FUNCTION_BLOCK Controller
  (* Standard: 61499-2 *)
  (* Version 0.1, 2015-00-21, Th?o, PC_THEO *)
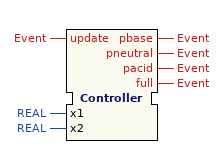
  EVENT_INPUT
    update;
  END_EVENT
  EVENT_OUTPUT
    pbase;
    pneutral;
    pacid;
    full;
  END_EVENT
  VAR_INPUT
    x1 : REAL;
    x2 : REAL;
  END_VAR
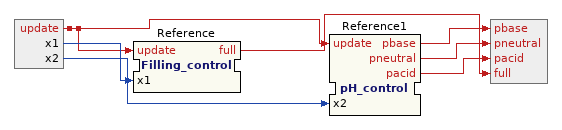
  FBS
    Reference : Filling_control;
    Reference1 : pH_control;
  END_FBS
  EVENT_CONNECTIONS
    update TO Reference.update;
    update TO Reference1.update;
    Reference1.pbase TO pbase;
    Reference1.pneutral TO pneutral;
    Reference1.pacid TO pacid;
    Reference.full TO full;
  END_CONNECTIONS
  DATA_CONNECTIONS
    x1 TO Reference.x1;
    x2 TO Reference1.x2;
  END_CONNECTIONS
END_FUNCTION_BLOCK
